(* CODESYS project CtaAppTime_1.0.0.1.library
   Description: Time Library der CTA
   Version: 1.0.0.1
   Title: CtaAppTime
   Author: SIS
   LanguageModelAttribute: qualified-access-only
   DocFormat: reStructuredText
   Placeholder: CtaAppTime
   DefaultNamespace: CtaAppTime
   CompiledLibraryCompatibilityVersion: CODESYS V3.5 SP16 Patch 3
   Company: CTA

Project tree, tasks and I/O mapping:
  libraries: VisuDialogs, * (System); VisuSymbols, 4.5.0.0 (System); CtaVisSymbols, 1.0.0.0 (CTA); CtaSysConfig, 1.0.0.2 (CTA); SysTime, 3.5.17.0 (System); Util, 3.5.19.0 (System); Standard, 3.5.18.0 (System); SysTypes Interfaces, * (System); CtaVisHelp, 1.0.0.0 (CTA)
  40 Visualizations/
    SCHEDULER/
      visualisation VIS_SCHEDULER_QUERY
      visualisation VIS_SCHEDULER_LINE
      visualisation VIS_SCHEDULER
      visualisation DIA_SCHEDULER_CONFIG
    INTERVALL/
      visualisation VIS_INTERVALL_LINE
      visualisation VIS_INTERVALL_QUERY
      visualisation VIS_INTERVALL
      visualisation DIA_INTERVALL_CONFIG
  30 Program Organization Units/
    function block fbTimeMeasurement [ST]: Start, Stop
    function block FB_SCHEDULER [ST]: CheckScheduler, actConfig, DEMANDE, WEEKDAY, ITF_P_Enable, ITF_P_WeekDay, ITF_P_StartTime, ITF_P_StopTime
    function block FB_INTERVALL [ST]: CheckTime, DEMANDE, REST_RUN, ITF_P_Enable, ITF_P_OnTime, ITF_P_OffTime, actConfig, RESTART_IN, PAUSE
    function FcWeekDay [ST]
    function FuGetLocalDateAndTime [ST]
    function FuGetDateAndTime [ST]
  00000000-0000-0000-0000-000000000000|D:\CoDeSys\LibrariesV3\trunk\Intern\CAA\CAA Template\3.4.0.0 draft\Placeholder.xml
  00000000-0000-0000-0000-000000000000|D:\CoDeSys\LibrariesV3\trunk\Intern\CAA\CAA Template\3.2.0.3 draft\Prefix.pdf
  00000000-0000-0000-0000-000000000000|D:\CoDeSys\LibrariesV3\trunk\Intern\CAA\CAA Template\3.5.2.0 draft\Placeholder.xml
  20 Structs/
    data type enWeekDay
    text list txtWeekDay
  50 Images/
  10 Documenation/
    global variables VersionHistory
    global variables readMe
  21 Interface/
    interface ITF_SCHEDULER: DEMANDE, WEEKDAY, ITF_P_Enable, ITF_P_WeekDay, ITF_P_StartTime, ITF_P_StopTime
    interface ITF_INTERVALL: RESTART_IN, REST_RUN, DEMANDE, ITF_P_Enable, ITF_P_OnTime, ITF_P_OffTime, PAUSE
  11 Library Parameter/
  12 Konstanten/
  60 Textlisten/
  13 Globale Variablen/
  text list GlobalTextList
*)

// 20 Structs/enWeekDay
{attribute 'qualified_only'}
TYPE enWeekDay :
(
	EVERY_DAY 			:= 0,
	MONDAY				:= 1,
	TUESDAY				:= 2,
	WEDNESDAY			:= 3,
	THURSDAY			:= 4,
	FRIDAY				:= 5,
	SATURDAY			:= 6,
	SUNDAY				:= 7,
	MONDAY_TO_FRIDAY	:= 8,
	WEEKEND				:= 9,
	FIRST_HALF_WEEK		:= 10,
	SEKON_HALF_WEEK		:= 11
);
END_TYPE

// 10 Documenation/VersionHistory
(* 

.. image:: ../../Images/CTA_Logo.jpg
   :align: right
   :width: 15% 

**Vorlage**   


============ =========== =========== ============================================
**Date**     **Version** **Author**  **Change**
------------ ----------- ----------- --------------------------------------------
04.03.2021   0.0.0.0     SIS         Vorlage erstellt

============ =========== =========== ============================================


*)
VAR_GLOBAL
    stInfo : STRING:= '0.0.0.0, Vorlage, CTA';
END_VAR

// 10 Documenation/readMe
(*

**ReadMe**

 
|	**Empfehlung**
|
|	Dokumentrieren Sie die Library für eine nachhaltige Entwicklung
|     
| *Beispiel*
| 
| Dies ist die Vorlage Library der CTA. Erstellen Sie ihre Library anhand dieser Vorlage.
*)

VAR_GLOBAL
    xReadMeDone              :   BOOL;
END_VAR

// 30 Program Organization Units/fbTimeMeasurement
FUNCTION_BLOCK fbTimeMeasurement 
VAR
    ltMessung   :   LTIME;    
END_VAR

METHOD Start 
VAR_INPUT
END_VAR
ltMessung := LTIME();
END_METHOD

METHOD Stop : LTIME
VAR_INPUT
END_VAR
Stop := LTIME() - ltMessung;
END_METHOD

END_FUNCTION_BLOCK

// 30 Program Organization Units/FB_SCHEDULER
FUNCTION_BLOCK FB_SCHEDULER IMPLEMENTS ITF_SCHEDULER
VAR_OUTPUT
	xDemande	:	BOOL;
END_VAR

VAR
	fbConfigFile		:	CtaSysConfig.fbConfigFile;
	fbxEnabele			:	CtaSysConfig.fbBOOL;
	fbenWeekDay			:	CtaSysConfig.fbINT;
	fbtodStart			:	CtaSysConfig.fbTOD;
	fbtodStop			:	CtaSysConfig.fbTOD;
END_VAR

actConfig();
CheckScheduler();

METHOD CheckScheduler
VAR_INPUT
END_VAR
VAR
	xCheckTime	:	BOOL;
	tdTemp		:	TOD;
END_VAR
xCheckTime := FALSE; 
IF fbxEnabele.proValue THEN
	IF fbenWeekDay.proValue = enWeekDay.EVERY_DAY THEN
		xCheckTime := TRUE;
	ELSIF fbenWeekDay.proValue = enWeekDay.MONDAY_TO_FRIDAY THEN
		IF FcWeekDay() <= Util.WEEKDAY.FRIDAY AND FcWeekDay()>= Util.WEEKDAY.MONDAY THEN
			xCheckTime := TRUE;
		ELSIF fbtodStart.proValue > fbtodStop.proValue THEN
			IF FcWeekDay() <= Util.WEEKDAY.SATURDAY THEN
				xCheckTime := TRUE;
			END_IF;
		ELSE
			xCheckTime := FALSE;	
		END_IF;
	ELSIF fbenWeekDay.proValue = enWeekDay.WEEKEND THEN
		IF FcWeekDay() >= Util.WEEKDAY.SATURDAY AND FcWeekDay() <= Util.WEEKDAY.SUNDAY THEN
			xCheckTime := TRUE;
		ELSE
			xCheckTime := FALSE;	
		END_IF;		
	ELSIF fbenWeekDay.proValue = enWeekDay.FIRST_HALF_WEEK THEN
		IF FcWeekDay() <= Util.WEEKDAY.WEDNESDAY THEN
			xCheckTime := TRUE;
		ELSIF fbtodStart.proValue > fbtodStop.proValue THEN
			IF FcWeekDay() <= Util.WEEKDAY.THURSDAY THEN
				xCheckTime := TRUE;
			END_IF;
		ELSE
			xCheckTime := FALSE;	
		END_IF;		
	ELSIF fbenWeekDay.proValue = enWeekDay.SEKON_HALF_WEEK THEN
		IF FcWeekDay() >= Util.WEEKDAY.THURSDAY THEN
			xCheckTime := TRUE;
		ELSE
			xCheckTime := FALSE;	
		END_IF;			
	ELSE
		IF fbenWeekDay.proValue = TO_INT(FcWeekDay()) THEN	
			xCheckTime := TRUE;
		ELSIF fbtodStart.proValue > fbtodStop.proValue THEN
			IF FcWeekDay() <> Util.WEEKDAY.SUNDAY THEN
				IF fbenWeekDay.proValue + 1 = FcWeekDay() THEN
					xCheckTime := TRUE;
				END_IF;
			ELSIF fbenWeekDay.proValue = enWeekDay.SUNDAY THEN
				IF FcWeekDay() = Util.WEEKDAY.MONDAY THEN
					xCheckTime := TRUE;
				END_IF;
			END_IF;
		ELSE
			xCheckTime := FALSE;
		END_IF;
	END_IF;
	
	IF xCheckTime THEN
		tdTemp := TO_TOD(FuGetLocalDateAndTime());
		IF tdTemp >= fbtodStart.proValue AND tdTemp <= fbtodStop.proValue THEN
			xDemande := TRUE;
		ELSE
			xDemande := FALSE;
		END_IF
	ELSE
		xDemande := FALSE;
	END_IF;
ELSE
	xDemande := FALSE;
END_IF;
END_METHOD

ACTION actConfig:
fbConfigFile();

fbxEnabele	(	_usiParaNr := 1,	itfConfigFb := fbConfigFile);
fbenWeekDay	(	_usiParaNr := 2,	itfConfigFb := fbConfigFile	,_MinInit	:= 0	,	_MaxInit	:= 11);
fbtodStart	(	_usiParaNr := 3,	itfConfigFb := fbConfigFile);
fbtodStop	(	_usiParaNr := 4,	itfConfigFb := fbConfigFile);
END_ACTION

PROPERTY DEMANDE : BOOL
GET
DEMANDE := xDemande;
END_GET
END_PROPERTY

PROPERTY WEEKDAY : enWeekDay
GET
WEEKDAY := fbenWeekDay.proValue;
END_GET
END_PROPERTY

PROPERTY ITF_P_Enable : CtaSysConfig.ITF_BOOL
GET
ITF_P_Enable := fbxEnabele;
END_GET
END_PROPERTY

PROPERTY ITF_P_WeekDay : CtaSysConfig.ITF_INT
GET
ITF_P_WeekDay := fbenWeekDay;
END_GET
END_PROPERTY

PROPERTY ITF_P_StartTime : CtaSysConfig.ITF_TOD
GET
ITF_P_StartTime := fbtodStart;
END_GET
END_PROPERTY

PROPERTY ITF_P_StopTime : CtaSysConfig.ITF_TOD
GET
ITF_P_StopTime := fbtodStop;
END_GET
END_PROPERTY

END_FUNCTION_BLOCK

// 21 Interface/ITF_SCHEDULER
INTERFACE ITF_SCHEDULER EXTENDS __SYSTEM.IQueryInterface

PROPERTY DEMANDE : BOOL
GET
END_GET
END_PROPERTY

PROPERTY WEEKDAY : enWeekDay
GET
END_GET
END_PROPERTY

PROPERTY ITF_P_Enable : CtaSysConfig.ITF_BOOL
GET
END_GET
END_PROPERTY

PROPERTY ITF_P_WeekDay : CtaSysConfig.ITF_INT
GET
END_GET
END_PROPERTY

PROPERTY ITF_P_StartTime : CtaSysConfig.ITF_TOD
GET
END_GET
END_PROPERTY

PROPERTY ITF_P_StopTime : CtaSysConfig.ITF_TOD
GET
END_GET
END_PROPERTY

END_INTERFACE

// 30 Program Organization Units/FcWeekDay
FUNCTION FcWeekDay : Util.WEEKDAY
VAR_INPUT
END_VAR
VAR
END_VAR

FcWeekDay := Util.DayOfWeek(TO_DATE(FuGetLocalDateAndTime()));

END_FUNCTION

// 30 Program Organization Units/FuGetLocalDateAndTime
FUNCTION FuGetLocalDateAndTime : DT
VAR_INPUT
END_VAR
VAR
	RTS_RESULT	:	SysTypes.RTS_IEC_RESULT;
	dwTemp		:	DWORD;
END_VAR

RTS_RESULT := SysTimeRtc.SysTimeRtcConvertUtcToLocal(SysTimeRtc.SysTimeRtcGet(RTS_RESULT),dwTemp);
FuGetLocalDateAndTime := TO_DT(dwTemp);

END_FUNCTION

// 30 Program Organization Units/FB_INTERVALL
FUNCTION_BLOCK FB_INTERVALL IMPLEMENTS ITF_INTERVALL
VAR_INPUT
	xReset		:	BOOL;
	xPause		:	BOOL;
END_VAR
VAR_OUTPUT
	xDemande	:	BOOL;
END_VAR

VAR
	tofOn				:	Standard.TOF;
	tofOff				:	Standard.TOF;
	tRestartIn			:	TIME;
	tRestTime			:	TIME;
	fbConfigFile		:	CtaSysConfig.fbConfigFile;
	fbxEnabele			:	CtaSysConfig.fbBOOL;
	fbtOn				:	CtaSysConfig.fbTIME;
	fbtOff				:	CtaSysConfig.fbTIME;
END_VAR

actConfig();
CheckTime();

METHOD CheckTime
VAR_INPUT
END_VAR
VAR
	xCheckTime	:	BOOL;
	tdTemp		:	TOD;
END_VAR
IF fbxEnabele.proValue THEN
	IF NOT xPause THEN
		IF NOT tofOn.Q OR fbtOn.proStateChanged THEN
			tofOn	(	IN	:= NOT tofOff.Q,PT	:= fbtOn.proValue);
		ELSE
			tofOn	(	IN	:= NOT tofOff.Q);
		END_IF;
		IF NOT tofOff.Q OR fbtOff.proStateChanged THEN
			tofOff	(	IN	:= tofOn.Q 	   ,PT	:= fbtOff.proValue);
		ELSE
			tofOff	(	IN	:= tofOn.Q 	   );
		END_IF;
		xDemande := tofOn.Q;
		IF xDemande THEN
			tRestartIn 	:= tofOn.PT - tofOn.ET + tofOff.PT;
			tRestTime	:= tofOn.PT - tofOn.ET;
		ELSE
			tRestartIn 	:= tofOff.PT - tofOff.ET;
			tRestTime 	:= T#0S;
		END_IF;
	ELSE
		tofOn	(	IN	:= tofOn.Q	,	PT	:= tRestTime);
		tofOff	(	IN	:= tofOff.Q ,	PT	:= tRestartIn-tRestTime);		
		xDemande 	:= FALSE;
	END_IF;
ELSE
	xDemande 	:= FALSE;
	tRestartIn 	:= T#0S;
	tRestTime 	:= T#0S;
END_IF;
IF fbxEnabele.proStateChanged THEN
	xReset := TRUE;
END_IF;
IF xReset THEN
	tofOn (IN := FALSE, PT := T#0S);
	tofOff(IN := FALSE, PT := T#0S);
	tRestTime	:= fbtOn.proValue;
	tRestartIn 	:= tRestTime + fbtOff.proValue;
	xReset := FALSE;
END_IF
END_METHOD

PROPERTY DEMANDE : BOOL
GET
DEMANDE := xDemande;
END_GET
END_PROPERTY

PROPERTY REST_RUN : TIME
GET
REST_RUN := tRestTime;
END_GET
END_PROPERTY

PROPERTY ITF_P_Enable : CtaSysConfig.ITF_BOOL
GET
ITF_P_Enable := fbxEnabele;
END_GET
END_PROPERTY

PROPERTY ITF_P_OnTime : CtaSysConfig.ITF_TIME
GET
ITF_P_OnTime := fbtOn;
END_GET
END_PROPERTY

PROPERTY ITF_P_OffTime : CtaSysConfig.ITF_TIME
GET
ITF_P_OffTime := fbtOff;
END_GET
END_PROPERTY

ACTION actConfig:
fbConfigFile();

fbxEnabele	(	_usiParaNr := 1,	itfConfigFb := fbConfigFile);
fbtOn		(	_usiParaNr := 2,	itfConfigFb := fbConfigFile);
fbtOff		(	_usiParaNr := 3,	itfConfigFb := fbConfigFile);

IF fbtOn.proMax > T#24D12H THEN
	fbtOn.proMax := T#24D12H;
END_IF;

IF fbtOff.proMax > T#24D12H THEN
	fbtOff.proMax := T#24D12H;
END_IF
END_ACTION

PROPERTY RESTART_IN : TIME
GET
RESTART_IN := tRestartIn;
END_GET
END_PROPERTY

PROPERTY PAUSE : BOOL
GET
PAUSE := xPause;
END_GET
END_PROPERTY

END_FUNCTION_BLOCK

// 21 Interface/ITF_INTERVALL
INTERFACE ITF_INTERVALL EXTENDS __SYSTEM.IQueryInterface

PROPERTY RESTART_IN : TIME
GET
END_GET
END_PROPERTY

PROPERTY REST_RUN : TIME
GET
END_GET
END_PROPERTY

PROPERTY DEMANDE : BOOL
GET
END_GET
END_PROPERTY

PROPERTY ITF_P_Enable : CtaSysConfig.ITF_BOOL
GET
END_GET
END_PROPERTY

PROPERTY ITF_P_OnTime : CtaSysConfig.ITF_TIME
GET
END_GET
END_PROPERTY

PROPERTY ITF_P_OffTime : CtaSysConfig.ITF_TIME
GET
END_GET
END_PROPERTY

PROPERTY PAUSE : BOOL
GET
END_GET
END_PROPERTY

END_INTERFACE

// 30 Program Organization Units/FuGetDateAndTime
FUNCTION FuGetDateAndTime : DT
VAR_INPUT
END_VAR
VAR
	RTS_RESULT	:	SysTypes.RTS_IEC_RESULT;
END_VAR

FuGetDateAndTime := TO_DT(TO_LINT(SysTimeRtc.SysTimeRtcGet(RTS_RESULT)));

END_FUNCTION

// 40 Visualizations/SCHEDULER/VIS_SCHEDULER_QUERY
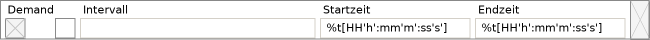
VISUALIZATION VIS_SCHEDULER_QUERY  // 650x40
VAR_INPUT
	ITF_SCHEDULER_IN		:	ITF_SCHEDULER;	
END_VAR
    Frame (0,0 650x40), invisible if: NOT __QUERYINTERFACE(ITF_SCHEDULER_IN,ITF_SCHEDULER_IN)
        shows VIS_SCHEDULER_LINE(ITF_SCHEDULER_IN := ITF_SCHEDULER_IN)
END_VISUALIZATION

// 40 Visualizations/SCHEDULER/VIS_SCHEDULER_LINE
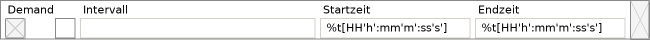
VISUALIZATION VIS_SCHEDULER_LINE  // 650x40
VAR_INPUT
	ITF_SCHEDULER_IN		:	ITF_SCHEDULER;	
END_VAR
    Image (5,18 20x20), image: CtaVisSymbols.ImagePool.close_red
    Textfield (80,18 235x20), text list: 'txtWeekDay', text index: ITF_SCHEDULER_IN.WEEKDAY
    Image (5,18 20x20), invisible if: NOT ITF_SCHEDULER_IN.DEMANDE, image: CtaVisSymbols.ImagePool.check_green
    Textfield (320,18 150x20), "%t[HH'h':mm'm':ss's']", text variable: ITF_SCHEDULER_IN.ITF_P_StartTime.proValue
    Textfield (475,18 150x20), "%t[HH'h':mm'm':ss's']", text variable: ITF_SCHEDULER_IN.ITF_P_StopTime.proValue
    Image (630,0 20x40), image: CtaVisSymbols.ImagePool.SettingsSmall
        OnMouseClick:  Dialog=DIA_SCHEDULER_CONFIG, Parameters={ITF_SCHEDULER_IN: ITF_SCHEDULER_IN}, OpenModal=True, OpenCentered=True
    Frame (55,18 20x20)
        shows CtaSysConfig.visBOOL(visfbBOOLIn := ITF_SCHEDULER_IN.ITF_P_Enable)
    Label (5,2 52x12), "Demand"
    Label (80,2 235x12), "Intervall"
    Label (320,2 115x12), "Startzeit"
    Label (475,2 150x12), "Endzeit"
END_VISUALIZATION

// 40 Visualizations/SCHEDULER/VIS_SCHEDULER
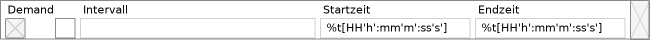
VISUALIZATION VIS_SCHEDULER  // 650x40
VAR_INPUT
	ITF_SCHEDULER_IN		:	ITF_SCHEDULER;	
END_VAR
    Frame (0,0 650x40), invisible if: NOT __QUERYINTERFACE(ITF_SCHEDULER_IN,ITF_SCHEDULER_IN)
        shows VIS_SCHEDULER_QUERY(ITF_SCHEDULER_IN := ITF_SCHEDULER_IN)
END_VISUALIZATION

// 40 Visualizations/INTERVALL/VIS_INTERVALL_LINE
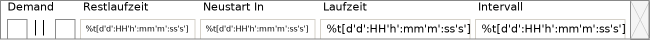
VISUALIZATION VIS_INTERVALL_LINE  // 650x40
VAR_INPUT
	ITF_INTERVALL_IN		:	ITF_INTERVALL;	
END_VAR
    Textfield (80,19 115x20), "%t[d'd':HH'h':mm'm':ss's']", text variable: ITF_INTERVALL_IN.REST_RUN
    Textfield (320,19 150x20), "%t[d'd':HH'h':mm'm':ss's']", text variable: ITF_INTERVALL_IN.ITF_P_OnTime.proValue
    Textfield (475,19 150x20), "%t[d'd':HH'h':mm'm':ss's']", text variable: ITF_INTERVALL_IN.ITF_P_OffTime.proValue
    Image (630,0 20x40), image: CtaVisSymbols.ImagePool.SettingsSmall
        OnMouseClick:  Dialog=DIA_INTERVALL_CONFIG, Parameters={ITF_INTERVALL_IN: ITF_INTERVALL_IN}, OpenModal=True, OpenCentered=True
    Frame (55,19 20x20)
        shows CtaSysConfig.visBOOL(visfbBOOLIn := ITF_INTERVALL_IN.ITF_P_Enable)
    Textfield (200,19 115x20), "%t[d'd':HH'h':mm'm':ss's']", text variable: ITF_INTERVALL_IN.RESTART_IN
    Line (35,20) (35,35), invisible if: NOT ITF_INTERVALL_IN.PAUSE
    Line (43,20) (43,35), invisible if: NOT ITF_INTERVALL_IN.PAUSE
    Label (5,2 52x10), "Demand"
    Label (80,2 115x10), "Restlaufzeit"
    Label (200,2 115x10), "Neustart In"
    Label (320,2 150x10), "Laufzeit"
    Label (475,2 150x10), "Intervall"
    Frame (7,19 20x20)
        shows CtaVisHelp.VIS_DI_Schalter(xDI := ITF_INTERVALL_IN.DEMANDE)
END_VISUALIZATION

// 40 Visualizations/INTERVALL/VIS_INTERVALL_QUERY
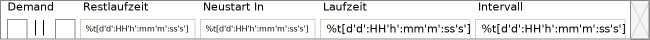
VISUALIZATION VIS_INTERVALL_QUERY  // 650x40
VAR_INPUT
	ITF_INTERVALL_IN		:	ITF_INTERVALL;	
END_VAR
    Frame (0,0 650x40), invisible if: NOT __QUERYINTERFACE(ITF_INTERVALL_IN,ITF_INTERVALL_IN)
        shows VIS_INTERVALL_LINE(ITF_INTERVALL_IN := ITF_INTERVALL_IN)
END_VISUALIZATION

// 40 Visualizations/INTERVALL/VIS_INTERVALL
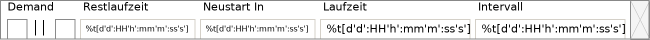
VISUALIZATION VIS_INTERVALL  // 650x40
VAR_INPUT
	ITF_INTERVALL_IN		:	ITF_INTERVALL;	
END_VAR
    Frame (0,0 650x40), invisible if: NOT __QUERYINTERFACE(ITF_INTERVALL_IN,ITF_INTERVALL_IN)
        shows VIS_INTERVALL_QUERY(ITF_INTERVALL_IN := ITF_INTERVALL_IN)
END_VISUALIZATION

// 40 Visualizations/INTERVALL/DIA_INTERVALL_CONFIG
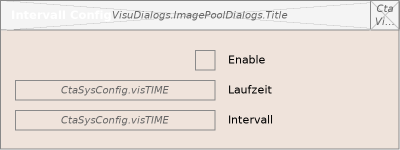
VISUALIZATION DIA_INTERVALL_CONFIG  // 400x150
VAR_INPUT
	ITF_INTERVALL_IN	:	ITF_INTERVALL;	
END_VAR
    Rectangle (0,0 399x149)
    Image (0,0 400x30), image: VisuDialogs.ImagePoolDialogs.Title
    Frame (195,50 20x20)
        shows CtaSysConfig.visBOOL(visfbBOOLIn := ITF_INTERVALL_IN.ITF_P_Enable)
    Frame (15,80 200x20)
        shows CtaSysConfig.visTIME(visfbTIMEIn := ITF_INTERVALL_IN.ITF_P_OnTime)
    Label (225,50 150x20), "Enable"
    Label (225,80 150x20), "Laufzeit"
    Label (225,110 150x20), "Intervall"
    Image (370,0 30x30), image: CtaVisSymbols.ImagePool.close_solo_black
        OnMouseClick:  Dialog=Current Dialog, Result=OK, NumpadKeypadSet=True
    Frame (15,110 200x20)
        shows CtaSysConfig.visTIME(visfbTIMEIn := ITF_INTERVALL_IN.ITF_P_OffTime)
    Label (0,0 150x30), "Intervall Config"
END_VISUALIZATION

// 40 Visualizations/SCHEDULER/DIA_SCHEDULER_CONFIG
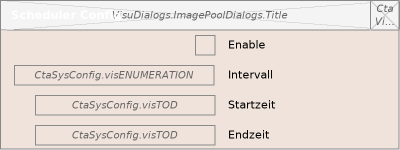
VISUALIZATION DIA_SCHEDULER_CONFIG  // 400x150
VAR_INPUT
	ITF_SCHEDULER_IN	:	ITF_SCHEDULER;	
END_VAR
    Rectangle (0,0 399x149)
    Image (0,0 400x30), image: VisuDialogs.ImagePoolDialogs.Title
    Frame (195,35 20x20)
        shows CtaSysConfig.visBOOL(visfbBOOLIn := ITF_SCHEDULER_IN.ITF_P_Enable)
    Label (225,35 150x20), "Enable"
    Label (225,95 150x20), "Startzeit"
    Label (225,125 150x20), "Endzeit"
    Image (370,0 30x30), image: CtaVisSymbols.ImagePool.close_solo_black
        OnMouseClick:  Dialog=Current Dialog, Result=OK, NumpadKeypadSet=True
    Frame (14,65 200x20), text list: 'txtWeekDay', text index: ITF_SCHEDULER_IN.ITF_P_WeekDay.proValue
        shows CtaSysConfig.visENUMERATION(visfbENUIn := ITF_SCHEDULER_IN.ITF_P_WeekDay)
    Label (225,65 150x20), "Intervall"
    Label (0,0 150x30), "Scheduler Config"
    Frame (35,95 180x20)
        shows CtaSysConfig.visTOD(visfbTODIn := ITF_SCHEDULER_IN.ITF_P_StartTime)
    Frame (35,125 180x20)
        shows CtaSysConfig.visTOD(visfbTODIn := ITF_SCHEDULER_IN.ITF_P_StopTime)
END_VISUALIZATION

(* text list txtWeekDay (id | default | de | en)
  0 | Täglich | Täglich | Every Day
  1 | Montag | Montag | Monday
  2 | Diensttag | Diensttag | Tuesday
  3 | Mittwoch | Mittwoch | Wednesday
  4 | Donnerstag | Donnerstag | Thursday
  5 | Freitag | Freitag | Friday
  6 | Samstag | Samstag | Saturday
  7 | Sonntag | Sonntag | Sunday
  8 | Mo-Fr | Mo-Fr | Mo-Fr
  9 | Wochenende | Wochenende | Weekend
  10 | Mo-Mi | Mo-Mi	 | Mo-Wed
  11 | Do-So | Do-So | Thu-Sun
   |  |  |  *)
